FUNCTION_BLOCK FB_Lamp_Test EXTENDS TcUnit.FB_TestSuite
VAR
	fbLamp : FB_Lamp;
	nExpected : BYTE;
	nResult : BYTE;
	bExpected : BOOL;
	bResult : BOOL;
END_VAR

TEST('Set bEnable TRUE');			 
fbLamp.bEnable := TRUE; 
fbLamp();
nExpected := 1;
nResult := fbLamp.GetControl();
AssertEquals(Expected := nExpected,
             Actual := nResult,
             Message := 'Control value is not correct');	 
TEST_FINISHED();

TEST('Set bEnable FALSE');			 
fbLamp.bEnable := FALSE; 
fbLamp();
nExpected := 0;
nResult := fbLamp.GetControl();
AssertEquals(Expected := nExpected,
             Actual := nResult,
             Message := 'Control value is not correct');	 
TEST_FINISHED();

END_FUNCTION_BLOCK

(* stored: Version 1.1.0.1, ProductVersion 3.1.4024.12
   POU FB_Lamp_Test: Id {174bf0a2-537b-03a1-3af1-2680370f6cfe}, SpecialFunc None *)
